RoboDK station: KUKAKR5.rdk

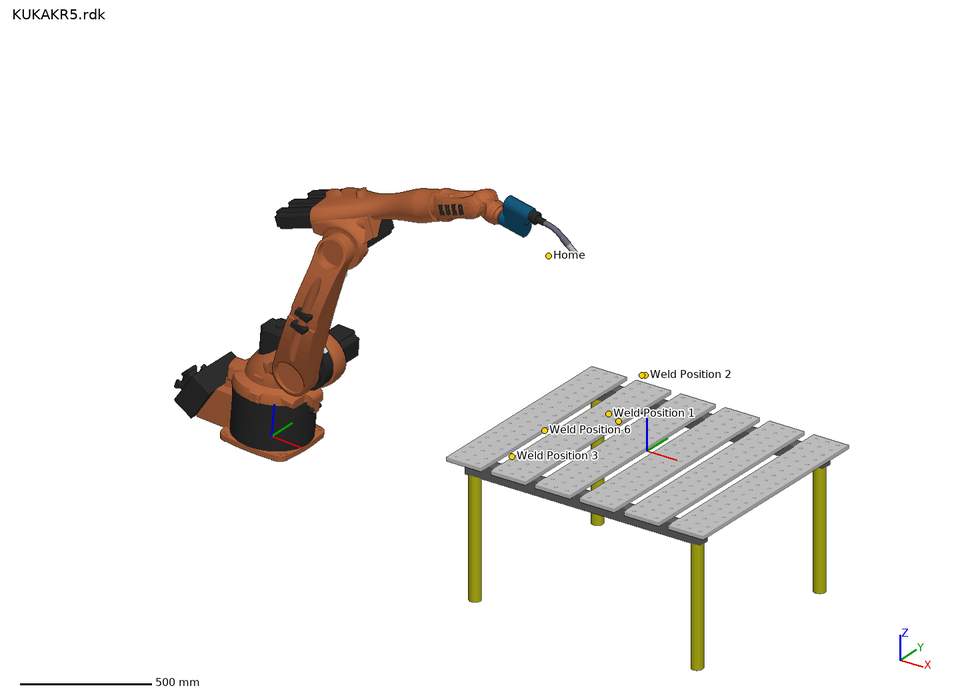
[picture v0: the station drawn from its stored meshes, robots at their saved joint values, targets as dots, program paths as lines]
Station KUKAKR5 (saved by RoboDK 5.7.1). Poses are relative to the parent item; angles as X-Y-Z fixed-axis rotations.
  - frame KUKA KR 5 arc Base at (-864.7, -362.92, 0) mm, rotated rx 0 ry 4.59 rz 0 deg
    - robot KUKA KR 5 arc: 6 axes, payload 5 kg, reach 1411 mm, repeatability 0.04 mm, weight 127 kg
        modified DH rows (alpha deg, a mm, theta deg, d mm): 0, 0, 0, 400; -90, 180, 0, 0; 0, 600, -90, 0; -90, 120, 0, 620; 90, 0, 0, 0; -90, 0, 180, 115
        joint limits [-155, -180, -15, -350, -130, -350] to [155, 65, 158, 350, 130, 350]; home [0, -90, 90, 0, 0, 0]; saved at [-0.53, -76.28, 54.78, 5.97, 27.95, -27.47]
      - tool Weld gun, TCP at (-4, 0, 371.3) mm, rotated rx 0 ry 45 rz 0 deg, size 299.9 x 60 x 318.3 mm
  - frame Frame 2 at (903.96, -397.16, 445.38) mm
    - object Object Table at (0, 0, 0) mm, size 1193.8 x 965.2 x 609.6 mm, geometry from Object Table.wrl
    - target Home  (Cartesian target) at (-482.36, 34.24, 678.62) mm, rotated rx -180 ry 45 rz -180 deg; joints [0, -90, 90, 0, 0, 0] of KUKA KR 5 arc
    - target Weld Position 1 (Cartesian target) at (-271.64, 131.05, 27.32) mm, rotated rx -180 ry 14.95 rz -176.3 deg; joints [-3.7, -59.95, 90, 0, 0, 0] of KUKA KR 5 arc
    - target Weld Position 2 (Cartesian target) at (-330.67, 457.46, 46.21) mm, rotated rx -180 ry 15.77 rz -163.6 deg; joints [-16.4, -60.77, 90, 0, 0, 0] of KUKA KR 5 arc
    - target Weld Position 3 (Cartesian target) at (-338.75, -415.51, 46.21) mm, rotated rx -180 ry 15.77 rz 162.54 deg; joints [17.46, -60.77, 90, 0, 0, 0] of KUKA KR 5 arc
    - target Weld Position 4 (Cartesian target) at (-149.25, 24.65, 74.96) mm, rotated rx 164.24 ry 39.27 rz 169.05 deg; joints [0.53, -56.68, 91.68, 1.19, -35.05, -13.14] of KUKA KR 5 arc
    - target Weld Position 5 (Cartesian target) at (-229.21, 291.53, 139.8) mm, rotated rx -152.08 ry 44.76 rz -127.37 deg; joints [0.53, -56.68, 91.68, 44.2, -52.8, -13.14] of KUKA KR 5 arc
    - target Weld Position 6 (Cartesian target) at (-256.28, -314.14, 140.91) mm, rotated rx -153.66 ry 44.13 rz -151.58 deg; joints [23.81, -57.5, 92.84, 44.2, -52.8, -15.53] of KUKA KR 5 arc
